TYPE ST_KNXnetIP_CommonHeader :
STRUCT
	nHeaderSize			: BYTE;
	nProtocolVersion	: BYTE;
	nServiceType		: WORD;
	nTotalLength		: WORD;
END_STRUCT
END_TYPE

(* stored: Version 1.1.0.1
   DUT ST_KNXnetIP_CommonHeader: Id {bed75fff-707e-49f6-ac0e-8d0050ddc958} *)
